Universal Robots PolyScope program: gravityFeederW.urp

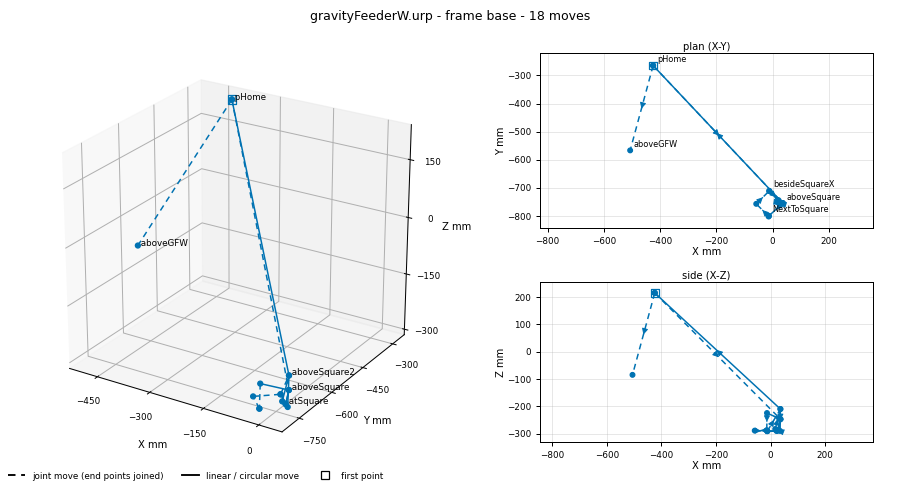
[picture p0: tool path of gravityFeederW.urp in frame base, 18 of 22 moves have a stored position in this frame; points joined in program order, loops and branches not executed]
Program gravityFeederW (installation=admin directory=/programs/WED_9AM createdIn=3.8.0.61336 lastSavedIn=3.15.8.106339 robotSerialNumber=2015350925)
Calibrated DH parameters: a=[0.000202, -0.047961, -0.392055, -0.000001, 0.000007, 0]; d=[0.089082, 828.736652, -823.627268, -4.999465, 0.094767, 0.082274]; alpha=[1.570325, 0.00051, -0.003464, 1.570175, -1.569769, 0]; deltaTheta=[0.000028, 1.457808, -1.502844, -6.238105, -6.283148, -0.000082]
Robot Program (runOnlyOnce=true)
  Set DigitalOutput pin=digital_out[0]; digitalValue=0
  Call _adminLinearIndex3
  Wait Sleep waitTime=1
  MoveJ speed 180 deg/s, acceleration 100 deg/s^2 (useActiveTCP=true)
    Waypoint pHome: TCP in base x=-424.656 y=-264.992 z=215.642 mm, rx=-1.1994 ry=-2.8936 rz=-0.0048 rad; joints [224.993, -90.01, -89.998, -90.011, 89.242, -0.022] deg; flange x=-423.067 y=-266.363 z=431.532 mm, rx=-1.1994 ry=-2.8936 rz=-0.0048 rad
    Waypoint aboveGFW: TCP in base x=-506.253 y=-566.61 z=-84.661 mm, rx=-1.1455 ry=-2.7528 rz=0.4317 rad; joints [238.433, -128.713, -90.876, -33.006, 85.231, 12.686] deg; flange x=-457.472 y=-520.856 z=120.619 mm, rx=-1.1455 ry=-2.7528 rz=0.4317 rad
  MoveL speed 250 mm/s, acceleration 1200 mm/s^2 (useActiveTCP=true) feature=GravityFeeder
    Waypoint atGFRel (Relative): relativeFromPosition TCP in base x=-506.246 y=-566.623 z=-84.635 mm, rx=-1.1455 ry=-2.7528 rz=0.4317 rad; joints [238.435, -128.711, -90.876, -33.006, 85.228, 12.688] deg; TCP in base x=-509.257 y=-572.851 z=-135.431 mm, rx=-1.1454 ry=-2.7521 rz=0.4332 rad; joints [238.505, -133.97, -90.585, -27.98, 85.21, 12.748] deg; pose in feature x=153.913 y=-140.7 z=-426.259 mm, rx=0.0087 ry=-3.1196 rz=-0.0475 rad; flange x=-460.302 y=-526.935 z=69.772 mm, rx=-1.1454 ry=-2.7521 rz=0.4332 rad
    Set DigitalOutput pin=digital_out[0]; digitalValue=1
    Wait Sleep waitTime=1
    Waypoint moveUpRel (Relative): motionParameters(jointSpeed=1.047198 jointAcceleration=1.396263 cartesianSpeed=0.02 cartesianAcceleration=0.02); relativeFromPosition TCP in base x=-509.785 y=-573.442 z=-137.41 mm, rx=-1.1452 ry=-2.7521 rz=0.4334 rad; joints [238.494, -134.234, -90.453, -27.841, 85.211, 12.728] deg; TCP in base x=-512.707 y=-576.409 z=-135.894 mm, rx=-1.1453 ry=-2.7522 rz=0.4335 rad; joints [238.41, -134.497, -89.605, -28.415, 85.242, 12.653] deg; pose in feature x=153.998 y=-145.203 z=-428.379 mm, rx=0.0088 ry=-3.1198 rz=-0.0473 rad; flange x=-463.747 y=-530.45 z=69.297 mm, rx=-1.1453 ry=-2.7522 rz=0.4335 rad
    Waypoint aboveGFRel (Relative): motionParameters(jointSpeed=1.047198 jointAcceleration=1.396263 cartesianSpeed=0.02 cartesianAcceleration=0.02); relativeFromPosition TCP in base x=-512.696 y=-576.419 z=-135.921 mm, rx=-1.1451 ry=-2.7523 rz=0.4335 rad; joints [238.41, -134.5, -89.604, -28.415, 85.245, 12.646] deg; TCP in base x=-506.118 y=-569.469 z=-121.514 mm, rx=-1.1454 ry=-2.7522 rz=0.4335 rad; joints [238.58, -132.21, -91.332, -28.993, 85.189, 12.82] deg; pose in feature x=153.912 y=-141.09 z=-411.602 mm, rx=0.0087 ry=-3.1198 rz=-0.0474 rad; flange x=-457.166 y=-523.52 z=83.682 mm, rx=-1.1454 ry=-2.7522 rz=0.4335 rad
  MoveJ speed 60 deg/s, acceleration 80 deg/s^2 (useActiveTCP=true)
    Waypoint pHome: TCP in base x=-424.656 y=-264.992 z=215.642 mm, rx=-1.1994 ry=-2.8936 rz=-0.0048 rad; joints [224.993, -90.01, -89.998, -90.011, 89.242, -0.022] deg; flange x=-423.067 y=-266.363 z=431.532 mm, rx=-1.1994 ry=-2.8936 rz=-0.0048 rad
    Waypoint aboveSquare: TCP in base x=36.387 y=-754.554 z=-247.163 mm, rx=1.2016 ry=2.8994 rz=-0.0037 rad; joints [281.141, -148.015, -74.126, -47.712, 89.943, 55.968] deg; flange x=35.974 y=-753.836 z=-31.264 mm, rx=1.2016 ry=2.8994 rz=-0.0037 rad
  MoveL speed 250 mm/s, acceleration 1200 mm/s^2 (useActiveTCP=true) feature=Base
    Waypoint atSquare: TCP in base x=27.975 y=-754.016 z=-286.557 mm, rx=1.2021 ry=2.8995 rz=-0.0036 rad; joints [280.522, -151.75, -73.506, -44.611, 89.942, 55.355] deg; flange x=27.617 y=-753.337 z=-70.659 mm, rx=1.2021 ry=2.8995 rz=-0.0036 rad
    Set DigitalOutput pin=digital_out[0]; digitalValue=0
    Wait Sleep waitTime=1
    Waypoint aboveSquare: TCP in base x=36.387 y=-754.554 z=-247.163 mm, rx=1.2016 ry=2.8994 rz=-0.0037 rad; joints [281.141, -148.015, -74.126, -47.712, 89.943, 55.968] deg; flange x=35.974 y=-753.836 z=-31.264 mm, rx=1.2016 ry=2.8994 rz=-0.0037 rad
    Waypoint NextToSquare: TCP in base x=-13.128 y=-799.041 z=-224.591 mm, rx=1.2019 ry=2.8993 rz=-0.0035 rad; joints [276.969, -151.009, -63.364, -55.49, 89.947, 51.825] deg; flange x=-13.559 y=-798.339 z=-8.693 mm, rx=1.2019 ry=2.8993 rz=-0.0035 rad
    Set DigitalOutput pin=digital_out[0]; digitalValue=1
    Wait Sleep waitTime=0.5
  MoveJ speed 180 deg/s, acceleration 100 deg/s^2 (useActiveTCP=true)
    Waypoint besideSquareY: TCP in base x=-13.979 y=-801.074 z=-288.268 mm, rx=1.2017 ry=2.8993 rz=-0.0034 rad; joints [276.893, -157.027, -61.628, -51.212, 89.962, 51.732] deg; flange x=-14.421 y=-800.39 z=-72.369 mm, rx=1.2017 ry=2.8993 rz=-0.0034 rad
  Wait Sleep waitTime=0.1
  MoveL speed 30 mm/s, acceleration 30 mm/s^2 (useActiveTCP=true) feature=Base
    If force()≤45 (checkContinuously=true)
      Waypoint atSquareY (Relative): relativeFromPosition TCP in base x=-13.971 y=-801.112 z=-288.239 mm, rx=1.2017 ry=2.8992 rz=-0.0035 rad; joints [276.893, -157.027, -61.624, -51.212, 89.963, 51.733] deg; TCP in base x=1.578 y=-785.719 z=-288.955 mm, rx=1.2018 ry=2.8992 rz=-0.0033 rad; joints [278.164, -155.29, -65.738, -48.838, 89.968, 52.999] deg; flange x=1.118 y=-785.041 z=-73.056 mm, rx=1.2018 ry=2.8992 rz=-0.0033 rad
    Wait Sleep waitTime=0.5
  MoveJ speed 180 deg/s, acceleration 100 deg/s^2 (useActiveTCP=true)
    Waypoint besideSquareY: TCP in base x=-13.979 y=-801.074 z=-288.268 mm, rx=1.2017 ry=2.8993 rz=-0.0034 rad; joints [276.893, -157.027, -61.628, -51.212, 89.962, 51.732] deg; flange x=-14.421 y=-800.39 z=-72.369 mm, rx=1.2017 ry=2.8993 rz=-0.0034 rad
    Waypoint linkingMove: motionParameters(blendRadius=0.005); TCP in base x=-58.166 y=-756.622 z=-289.108 mm, rx=1.2018 ry=2.8995 rz=-0.0034 rad; joints [273.941, -152.445, -72.394, -45.037, 89.973, 48.766] deg; flange x=-58.56 y=-755.949 z=-73.21 mm, rx=1.2018 ry=2.8995 rz=-0.0034 rad
    Waypoint besideSquareX: TCP in base x=-11.874 y=-710.677 z=-291.242 mm, rx=1.2017 ry=2.8995 rz=-0.0033 rad; joints [277.95, -148.186, -83.128, -38.559, 89.981, 52.757] deg; flange x=-12.29 y=-710.014 z=-75.343 mm, rx=1.2017 ry=2.8995 rz=-0.0033 rad
  Wait Sleep waitTime=0.1
  MoveL speed 30 mm/s, acceleration 30 mm/s^2 (useActiveTCP=true) feature=Base
    If force()≤45 (checkContinuously=true)
      Waypoint atSquareX: TCP in base x=21.957 y=-744.876 z=-290.622 mm, rx=1.2021 ry=2.8994 rz=-0.0033 rad; joints [280.187, -151.247, -75.553, -43.073, 89.958, 55.016] deg; flange x=21.56 y=-744.226 z=-74.723 mm, rx=1.2021 ry=2.8994 rz=-0.0033 rad
    Wait Sleep waitTime=0.5
  MoveJ speed 60 deg/s, acceleration 80 deg/s^2 (useActiveTCP=true)
    Waypoint besideSquareX: TCP in base x=-11.874 y=-710.677 z=-291.242 mm, rx=1.2017 ry=2.8995 rz=-0.0033 rad; joints [277.95, -148.186, -83.128, -38.559, 89.981, 52.757] deg; flange x=-12.29 y=-710.014 z=-75.343 mm, rx=1.2017 ry=2.8995 rz=-0.0033 rad
    Waypoint aboveSquare2: TCP in base x=36.038 y=-754.121 z=-209.989 mm, rx=1.2012 ry=2.8998 rz=-0.0034 rad; joints [281.12, -144.584, -74.474, -50.811, 89.931, 55.933] deg; flange x=35.647 y=-753.459 z=5.91 mm, rx=1.2012 ry=2.8998 rz=-0.0034 rad
    Set DigitalOutput pin=digital_out[0]; digitalValue=0
    Wait Sleep waitTime=1
  MoveL speed 250 mm/s, acceleration 1200 mm/s^2 (useActiveTCP=true) feature=Base
    Waypoint atSquare2: TCP in base x=34.929 y=-756.694 z=-290.333 mm, rx=1.2013 ry=2.8997 rz=-0.0033 rad; joints [281.004, -152.426, -72.693, -44.749, 89.951, 55.806] deg; flange x=34.531 y=-756.032 z=-74.435 mm, rx=1.2013 ry=2.8997 rz=-0.0033 rad
    Set DigitalOutput pin=digital_out[0]; digitalValue=1
    Wait Sleep waitTime=1
    Waypoint easeout: TCP in base x=16.999 y=-751.256 z=-283.255 mm, rx=1.2013 ry=2.8997 rz=-0.0032 rad; joints [279.722, -151.117, -74.307, -44.451, 89.958, 54.524] deg; flange x=16.598 y=-750.614 z=-67.356 mm, rx=1.2013 ry=2.8997 rz=-0.0032 rad
    Waypoint aboveSquare2: TCP in base x=36.038 y=-754.121 z=-209.989 mm, rx=1.2012 ry=2.8998 rz=-0.0034 rad; joints [281.12, -144.584, -74.474, -50.811, 89.931, 55.933] deg; flange x=35.647 y=-753.459 z=5.91 mm, rx=1.2012 ry=2.8998 rz=-0.0034 rad
  MoveL speed 250 mm/s, acceleration 1200 mm/s^2 (useActiveTCP=true) feature=Base
    Waypoint pHome: TCP in base x=-424.656 y=-264.992 z=215.642 mm, rx=-1.1994 ry=-2.8936 rz=-0.0048 rad; joints [224.993, -90.01, -89.998, -90.011, 89.242, -0.022] deg; flange x=-423.067 y=-266.363 z=431.532 mm, rx=-1.1994 ry=-2.8936 rz=-0.0048 rad
SubProgram -> _adminLinearIndex3
SubProgram _adminLinearIndex3 (keepSynchronizedWithDisk=false) programFile=/programs/me345_admin/_adminLinearIndex3.urp
  Folder Move_linear_slide_Index3
    var_1 := False
    Loop While (checkContinuously=false) expression=var_1≟ False
      var_1 := socket_open("10.241.34.48",4001)
    var_3 := 1
    Send := "s r0x24 21"
    Script: socket_send_string(Send)
    Script: socket_send_byte(13)
    Send_Reply := socket_read_string()
    Send := "s r0xca 112778"
    Script: socket_send_string(Send)
    Script: socket_send_byte(13)
    Send_Reply := socket_read_string()
    Send := "t 1"
    Script: socket_send_string(Send)
    Script: socket_send_byte(13)
    Send_Reply := socket_read_string()
    Loop While (checkContinuously=false) expression=var_3≠0
      Send := "g r0xA0"
      Script: socket_send_string(Send)
      Script: socket_send_byte(13)
      var_3 := socket_get_var("v")
      Wait Sleep waitTime=0.1
    Script: socket_close()
    Script: sync()
